INTERFACE IMQTTMsgDecoder

METHOD decode : BOOL
VAR_INPUT
	Topic		: REFERENCE TO STRING;
	Data		: REFERENCE TO STRING;
END_VAR
END_METHOD

END_INTERFACE

(* stored: Version 1.1.0.1
   Itf IMQTTMsgDecoder: Id {74b1eb81-11fe-080f-1461-71298c8b3a2a}
   Method decode: Id {ba8ead04-d4c2-0f63-372d-bb025f22cbe2} *)
